// TIA Portal V19 export
TYPE "SpeedMachine_Alr"
// stored: Access Published
   STRUCT
      BrakeTimeOut : Bool;
      S120_ComErr : Bool;
      Ax : Struct
         Drive { ExternalAccessible := 'False'; ExternalVisible := 'False'; ExternalWritable := 'False'} : Bool;
      END_STRUCT;
      Fan_M : "MotorAlr";
   END_STRUCT;
END_TYPE
